# EPICS IOC start-up script: iocsh/iocStats-host.iocsh
dbLoadRecords("iocAdminSoft-freia-host.db", "IOC=$(HOSTNAME)")
